(* Logix 5000 project; controller HP_SSC01 vendor 1 type 14 code 67 rev 17.7; software revision 17.01; part 15 of 15 *)
(* tags used below, declared in another part *)
   A_C3_0200 : ALIAS FOR S_C3_FaultSafety.0;
   A_C3_0201 : ALIAS FOR S_C3_FaultSafety.1;
   A_C3_0202 : ALIAS FOR S_C3_FaultSafety.2;
   A_C3_0203 : ALIAS FOR S_C3_FaultSafety.3;
   A_C3_0204 : ALIAS FOR S_C3_FaultSafety.4;
   A_C3_0206 : ALIAS FOR S_C3_FaultSafety.6;
   A_C3_0208 : ALIAS FOR S_C3_FaultSafety.8;
   A_C3_0209 : ALIAS FOR S_C3_FaultSafety.9;
   A_C3_0210 : ALIAS FOR S_C3_FaultSafety.10;
   A_C3_0211 : ALIAS FOR S_C3_FaultSafety.11;
   A_C3_0216 : ALIAS FOR S_C3_FaultSafety.16;
   A_C3_0217 : ALIAS FOR S_C3_FaultSafety.17;
   A_C3_0220 : ALIAS FOR S_C3_FaultSafety.20;
   A_S01_0104 : ALIAS FOR System_FaultSafeIO.4;
   A_S01_0122 : ALIAS FOR System_FaultSafeIO.22;
   C3_EvacInPositionTest : DINT;
   RCS_CMD_EvacToStation : BOOL;
   RCS_SafeMemory_S01 : Udt_RCS_SafeData;
   RCS_SyncMotionEnable : BOOL;
   S_C3_AtEvacSpeed : BOOL;
   S_C3_BrakeTest : BOOL;
   S_C3_DumpTest : BOOL;
   S_C3_EvacOK : BOOL;
   S_C3_FaultReset : BOOL;
   S_C3_FaultSafety : DINT;
   S_C3_FaultSafety_OK : BOOL;
   S_C3_FaultStandard : DINT;
   S_C3_FaultStandard_OK : BOOL;
   S_C3_FW_LocalOK : BOOL;
   S_C3_InEvacPosition : BOOL;
   S_C3_MaintEnable : BOOL;
   S_C3_MCC3_LIM_MCR : ALIAS FOR C3_Safe:O.Pt04Data;
   S_C3_ModeLocal : BOOL;
   S_C3_ModeRemote : BOOL;
   S_C3_MotionEnabled : BOOL;
   S_C3_MotorActualPositionX1000 : DINT;
   S_C3_MotorAverageVelocityX1000 : DINT;
   S_C3_MSTOP_A : ALIAS FOR C3_Safe:I.Pt06Data;
   S_C3_MSTOP_B : ALIAS FOR C3_Safe:I.Pt07Data;
   S_C3_MSTOP_LT : ALIAS FOR C3_Safe:O.Pt02Data;
   S_C3_OIT_FaultReset : BOOL;
   S_C3_ONS : DINT;
   S_C3_ONS_Status : BOOL;
   S_C3_OutputEnable : BOOL;
   S_C3_PressureOK : ALIAS FOR C3_Safe:I.Pt05Data;
   S_C3_ResetTOF : TIMER;
   S_C3_SAFE_OFF_FDBK1 : ALIAS FOR C3_Safe:I.Pt01Data;
   S_C3_SAFE_OFF_FDBK2 : ALIAS FOR C3_Safe:I.Pt00Data;
   S_C3_SafeOff_ROUT : REDUNDANT_OUTPUT;
   S_C3_SAFETY_ENABLE_1 : ALIAS FOR C3_Safe:O.Pt00Data;
   S_C3_SAFETY_ENABLE_2 : ALIAS FOR C3_Safe:O.Pt01Data;
   S_C3_SS_RemoteMode : BOOL;
   S_C3_Stop0_OK : BOOL;
   S_C3_Stop1_OK : BOOL;
   S_C3_Stop1_OK_TOF : TIMER;
   S_FlashOn : TIMER;
   S_RCS_CMD_FaultReset : BOOL;
   S_RCS_MotionEnable : BOOL;
   S_System_FaultStandard : DINT;
   SSC_Stop0_OK : BOOL;
   SSC_Stop1_OK : BOOL;
(* SafeCarousel3, continued *)

ROUTINE SC335_SafetyOutputs   (* ladder *)
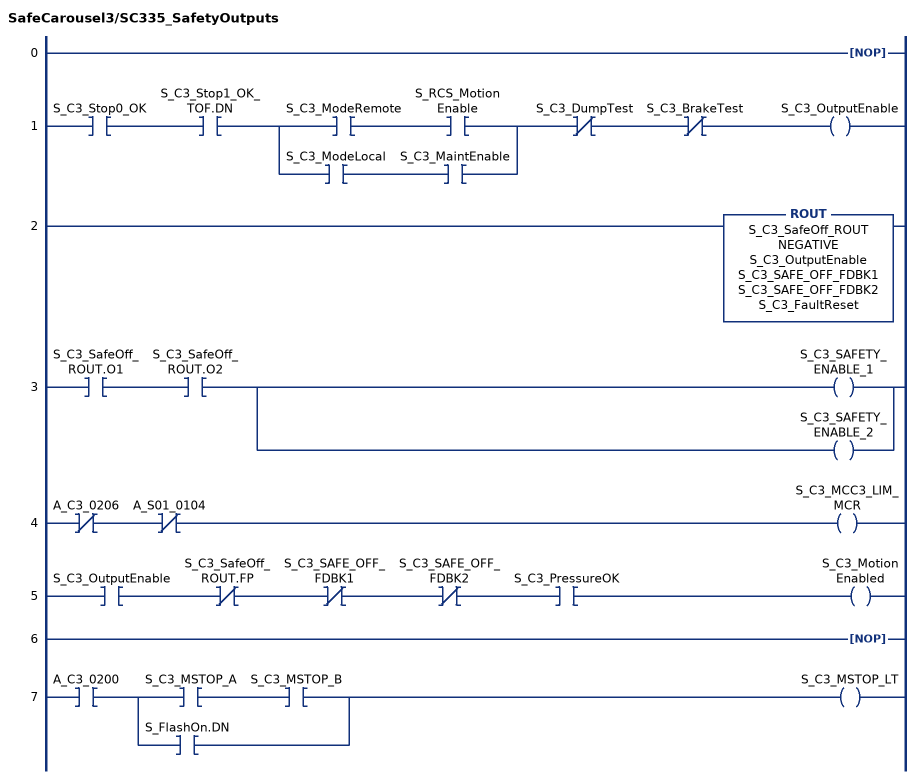
   0: NOP();
   1: XIC(S_C3_Stop0_OK)XIC(S_C3_Stop1_OK_TOF.DN)[XIC(S_C3_ModeRemote) XIC(S_RCS_MotionEnable) ,XIC(S_C3_ModeLocal) XIC(S_C3_MaintEnable) ]XIO(S_C3_DumpTest)XIO(S_C3_BrakeTest)OTE(S_C3_OutputEnable);
   2: ROUT(S_C3_SafeOff_ROUT,NEGATIVE,S_C3_OutputEnable,S_C3_SAFE_OFF_FDBK1,S_C3_SAFE_OFF_FDBK2,S_C3_FaultReset);
   3: XIC(S_C3_SafeOff_ROUT.O1)XIC(S_C3_SafeOff_ROUT.O2)[OTE(S_C3_SAFETY_ENABLE_1) ,OTE(S_C3_SAFETY_ENABLE_2) ];
   4: XIO(A_C3_0206)XIO(A_S01_0104)OTE(S_C3_MCC3_LIM_MCR);
   5: XIC(S_C3_OutputEnable)XIO(S_C3_SafeOff_ROUT.FP)XIO(S_C3_SAFE_OFF_FDBK1)XIO(S_C3_SAFE_OFF_FDBK2)XIC(S_C3_PressureOK)OTE(S_C3_MotionEnabled);
   6: NOP();
   7: XIC(A_C3_0200)[XIC(S_C3_MSTOP_A) XIC(S_C3_MSTOP_B) ,XIC(S_FlashOn.DN) ]OTE(S_C3_MSTOP_LT);
END_ROUTINE

ROUTINE SC340_Status   (* ladder *)
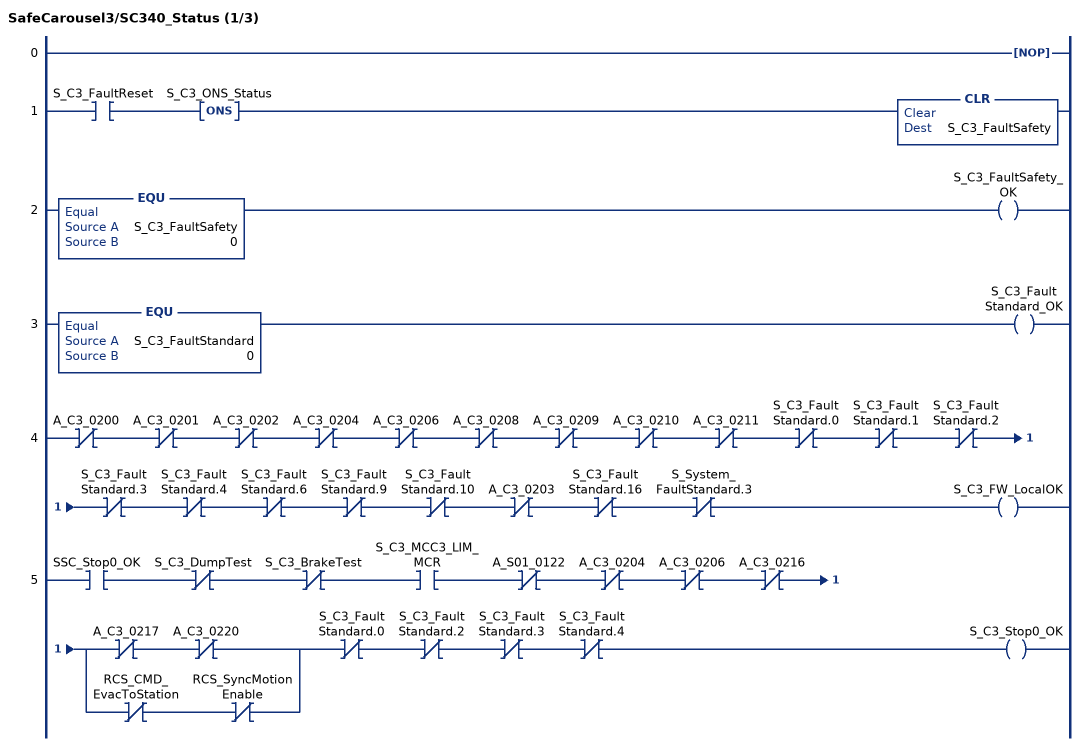
   0: NOP();
   1: XIC(S_C3_FaultReset)ONS(S_C3_ONS_Status)CLR(S_C3_FaultSafety);
   2: EQU(S_C3_FaultSafety,0)OTE(S_C3_FaultSafety_OK);
   3: EQU(S_C3_FaultStandard,0)OTE(S_C3_FaultStandard_OK);
   4: XIO(A_C3_0200)XIO(A_C3_0201)XIO(A_C3_0202)XIO(A_C3_0204)XIO(A_C3_0206)XIO(A_C3_0208)XIO(A_C3_0209)XIO(A_C3_0210)XIO(A_C3_0211)XIO(S_C3_FaultStandard.0)XIO(S_C3_FaultStandard.1)XIO(S_C3_FaultStandard.2)XIO(S_C3_FaultStandard.3)XIO(S_C3_FaultStandard.4)XIO(S_C3_FaultStandard.6)XIO(S_C3_FaultStandard.9)XIO(S_C3_FaultStandard.10)XIO(A_C3_0203)XIO(S_C3_FaultStandard.16)XIO(S_System_FaultStandard.3)OTE(S_C3_FW_LocalOK);
   5: XIC(SSC_Stop0_OK)XIO(S_C3_DumpTest)XIO(S_C3_BrakeTest)XIC(S_C3_MCC3_LIM_MCR)XIO(A_S01_0122)XIO(A_C3_0204)XIO(A_C3_0206)XIO(A_C3_0216)[XIO(A_C3_0217) XIO(A_C3_0220) ,XIO(RCS_CMD_EvacToStation) XIO(RCS_SyncMotionEnable) ]XIO(S_C3_FaultStandard.0)XIO(S_C3_FaultStandard.2)XIO(S_C3_FaultStandard.3)XIO(S_C3_FaultStandard.4)OTE(S_C3_Stop0_OK);
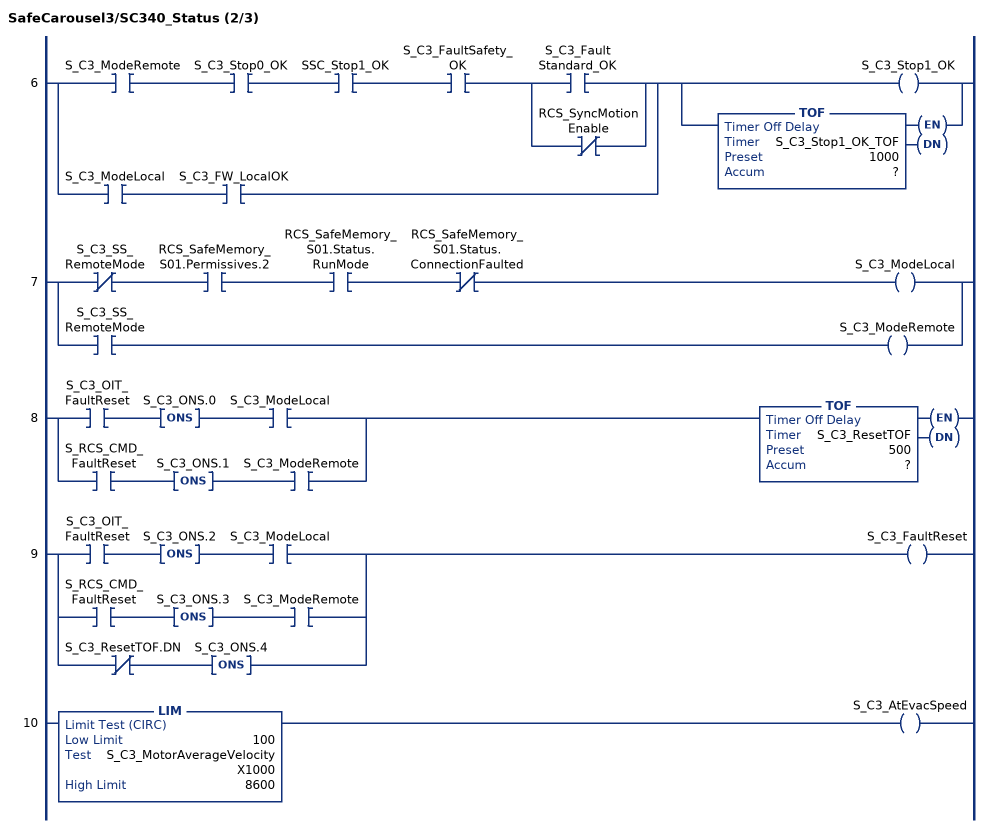
   6: [XIC(S_C3_ModeRemote) XIC(S_C3_Stop0_OK) XIC(SSC_Stop1_OK) XIC(S_C3_FaultSafety_OK) [XIC(S_C3_FaultStandard_OK) ,XIO(RCS_SyncMotionEnable) ] ,XIC(S_C3_ModeLocal) XIC(S_C3_FW_LocalOK) ][OTE(S_C3_Stop1_OK) ,TOF(S_C3_Stop1_OK_TOF,?,?) ];
   7: [XIO(S_C3_SS_RemoteMode) XIC(RCS_SafeMemory_S01.Permissives.2) XIC(RCS_SafeMemory_S01.Status.RunMode) XIO(RCS_SafeMemory_S01.Status.ConnectionFaulted) OTE(S_C3_ModeLocal) ,XIC(S_C3_SS_RemoteMode) OTE(S_C3_ModeRemote) ];
   8: [XIC(S_C3_OIT_FaultReset) ONS(S_C3_ONS.0) XIC(S_C3_ModeLocal) ,XIC(S_RCS_CMD_FaultReset) ONS(S_C3_ONS.1) XIC(S_C3_ModeRemote) ]TOF(S_C3_ResetTOF,?,?);
   9: [XIC(S_C3_OIT_FaultReset) ONS(S_C3_ONS.2) XIC(S_C3_ModeLocal) ,XIC(S_RCS_CMD_FaultReset) ONS(S_C3_ONS.3) XIC(S_C3_ModeRemote) ,XIO(S_C3_ResetTOF.DN) ONS(S_C3_ONS.4) ]OTE(S_C3_FaultReset);
   10: LIM(100,S_C3_MotorAverageVelocityX1000,8600)OTE(S_C3_AtEvacSpeed);
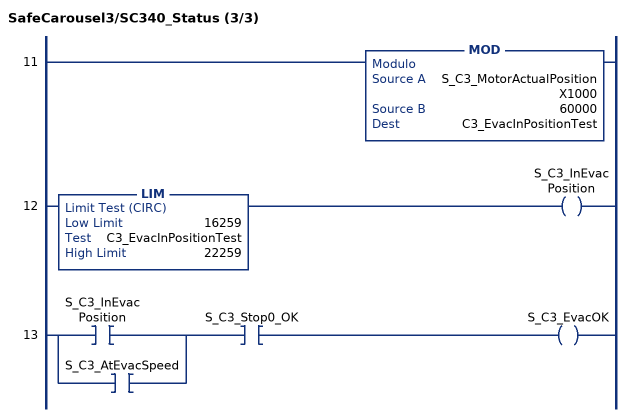
   11: MOD(S_C3_MotorActualPositionX1000,60000,C3_EvacInPositionTest);
   12: LIM(16259,C3_EvacInPositionTest,22259)OTE(S_C3_InEvacPosition);
   13: [XIC(S_C3_InEvacPosition) ,XIC(S_C3_AtEvacSpeed) ]XIC(S_C3_Stop0_OK)OTE(S_C3_EvacOK);
END_ROUTINE
END_PROGRAM
